// TIA Portal V17 export
GraphicList "Codex_GraphicList_Empty"  ListRange=Decimal, Comment="Codex empty graphic list import/export loop test."
